PROGRAM prgComEffIO
VAR
	fbCom		: FB_MqttCommunicator_v3;

END_VAR

fbCom(
	bConnect:= TRUE, 
	strAuthkey := 'DEV01673741737',
	sUserName:= '15410e61-b610-45b5-8f44-ee3f7b94538f' , 		
	sUserPassword:= 'c2948af7-82b2-4c6a-bb6c-453826157d1f',
	eSavePositionCertificate:= eSavePositionOnPLC.ePostionC, 
	bConnected=> , 
	bError=> , 
	hrErrorCode=> , 
	eConnectionState=> , 
	eErrorMessage_Out=> );

END_PROGRAM

(* stored: Version 1.1.0.1, ProductVersion 3.1.4024.12
   POU prgComEffIO: Id {cbcd318b-bf51-484c-bcaa-d6efcdf43fe3}, SpecialFunc None *)
